FUNCTION F_SAFETY_StatusFB_TO_RS : ST_SAFETY_FBRS
VAR_INPUT
	stFBStatus						: ST_SAFETY_FBStatus; 	(* Struktura ogolna *)
END_VAR

F_SAFETY_StatusFB_TO_RS.uStatus.stStatusWords 		:= stFBStatus;									(* Przepisanie *)
F_SAFETY_StatusFB_TO_RS.eState					 	:= stFBStatus.BState;							(* Ustawienie enum *)

END_FUNCTION

(* stored: Version 1.1.0.1, ProductVersion 3.1.4022.12
   POU F_SAFETY_StatusFB_TO_RS: Id {6071a81b-fb55-4442-8493-3a94bb1dac9e}, SpecialFunc None *)
